TYPE teCTCHomeMode :
(
	CTC_HOME_MODE_DIRECT 		:= 0,
	CTC_HOME_MODE_ENDSTOPIN 	:= 1,
	CTC_HOME_MODE_ENDSTOPOUT 	:= 2
);
END_TYPE

(* stored: Version 1.1.0.1, ProductVersion 3.1.4026.17
   EnumerationTextList teCTCHomeMode: Id {c5bbb05f-1f68-4c70-a2c3-31d4849b7196} *)
